// TIA Portal V21 export
VAR_GLOBAL   // PLC tag table "Default tag table"
   test AT %Q0.0 : Bool;
END_VAR
